FUNCTION_BLOCK ActMove
VAR_INPUT
END_VAR
VAR_OUTPUT
END_VAR
VAR
END_VAR

// NETWORK 1

END_FUNCTION_BLOCK

(* stored: Version 1.1.0.1, ProductVersion 3.1.4020.12
   POU ActMove: Id {20bb0f8e-cdc2-4082-aff9-51f6a4e205d9}, SpecialFunc None *)
